# B&R Automation Studio project SiemensBRCommunication (part 2)

#### DAVclient.st - Services communcations between a B&R and Siemens PLC
```iecst
(********************************************************************************************************************************)
(* COPYRIGHT -- B&R Industrial Automation																																												*)
(********************************************************************************************************************************)
(* Library:				DAVNoDave																																																			*)
(* File: 					DAVclient.st																																																	*)
(* Author: 				morrisd																																																				*)
(* Created: 			June 02, 2009																																																	*)
(********************************************************************************************************************************)

(********************************************************************************************************************************)
(* DAVclient																																																										*)
(*==============================================================================================================================*)
(* Services communications between the PLC and the Siemen's PLC																																	*)
(* Returns a status																																																							*)
(********************************************************************************************************************************)
FUNCTION_BLOCK DAVclient

	(* Function not enabled *)
	IF(enable = FALSE)THEN
		status:= 65534;

	(* Invalid handle *)
	ELSIF(pHandle = 0)THEN
 		status:= DAV_ERR_HANDLE;

	(* Run the function *)
	ELSE
		(* Make status busy *)
		status:= 65535;

		(****************************************************************************************************************************)
		(* Initialize function																									                  																	*)
		(****************************************************************************************************************************)
		IF(state = 0)THEN
			pDAV ACCESS pHandle;																	(* Access handle *)

			(* Valid configuration 0 *)
			IF(pDAV.internal = 2)THEN
				pDAV.internal:= 3;

				(* Initialize DAVsend *)
				memset(ADR(DAVexchange_0), 0, SIZEOF(DAVexchange_0));
				DAVexchange_0.enable:=						TRUE;							(* Enable function block *)
				DAVexchange_0.pHandle:=						pHandle;					(* Handle from DAVinitialize *)
				DAVexchange_0.sendLength:=				0;								(* Size of sending data - calculated later *)
				DAVexchange_0.timeout:=						timeout;					(* Pass timeout *)
				DAVexchange_0.mpiFullExchange:=	 TRUE;							(* Enable full exchange of data *)

				(* Check initialization *)
				IF((pDAV.pBufferR <> 0) AND (pDAV.pBufferW <> 0) AND (pDAV.pConfig <> 0) AND (pDAV.pMapping <> 0) AND (pDAV.maxLinesMapping > 0))THEN

					(* Clear the internal variables *)
					IF(pDAV.maxLinesConfig > 0)THEN
						FOR itemIdx:=0 TO pDAV.maxLinesConfig-1 BY 1 DO
							pConfig ACCESS pDAV.pConfig + (itemIdx * SIZEOF(pConfig));
							pConfig.internal:= 0;
						END_FOR
					END_IF
					IF(pDAV.maxLinesMapping > 0)THEN
						FOR itemIdx:=0 TO pDAV.maxLinesMapping-1 BY 1 DO
							pMapping ACCESS pDAV.pMapping + (itemIdx * SIZEOF(pMapping));
							pMapping.internal:= 0;
						END_FOR
					END_IF
					itemIdx:= 0;																			(* Reset looping index *)
					state:= 2;																				(* Start function block - READ all WRITE data *)

				(* Connection closed *)
				ELSIF(pDAV.internal = 1)THEN
					status:= DAV_ERR_CONNECT_CLOSED;

				(* Critical error *)
				ELSE
					status:= DAV_ERR_INITIALIZATION;
				END_IF

			(* Critical error *)
			ELSE
				status:= DAV_ERR_INITIALIZATION;
			END_IF
		END_IF
		(****************************************************************************************************************************)

		(****************************************************************************************************************************)
		(* Request to initialize the client																																													*)
		(* Note: code placed underneath STATE 0, to ensure pDAV is a valid pointer																									*)
		(****************************************************************************************************************************)
		IF((pDAV.internal = 2) OR (
			(pDAV.connection.protocol <> DAV_PROTOCOL_TCP) AND (pDAV.connection.protocol <> DAV_PROTOCOL_MPI)) )THEN
			errorPackets:= 0;																			(* Clear number of error packets *)
			state:= 0;																						(* Reset function block *)
		END_IF
		(****************************************************************************************************************************)

		(****************************************************************************************************************************)
		(* Pause and Resume the function block                                                   																		*)
		(****************************************************************************************************************************)
		IF((pause = TRUE) AND (state = 1))THEN
			state:= 254;																					(* Pause function block *)
		END_IF
		IF((pause = FALSE) AND (state = 254))THEN
			state:= 1;																						(* Resume function block *)
		END_IF
		paused:= (state = 254);																	(* Show PAUSE status *)
		(****************************************************************************************************************************)

		(****************************************************************************************************************************)
		(* Completed reading all WRITE variables                                                																		*)
		(****************************************************************************************************************************)
		IF((state = 2) AND (itemIdx >= pDAV.maxLinesMapping))THEN

 			(* Clear the internal variables *)
			IF(pDAV.maxLinesConfig > 0)THEN
				FOR itemIdx:=0 TO pDAV.maxLinesConfig-1 BY 1 DO
					pConfig ACCESS pDAV.pConfig + (itemIdx * SIZEOF(pConfig));
					pConfig.internal:= 0;
				END_FOR
			END_IF

			(* Clear the internal variables *)
			IF(pDAV.maxLinesMapping > 0)THEN
				FOR itemIdx:=0 TO pDAV.maxLinesMapping-1 BY 1 DO
					pMapping ACCESS pDAV.pMapping + (itemIdx * SIZEOF(pMapping));
					pMapping.internal:= 0;
				END_FOR
			END_IF

			itemIdx:= 0;																					(* Reset looping index *)
			currentPriority:= 1;																	(* Reset the prioirty *)
			currentMode:= 0;																			(* Set mode to WRITE *)
			state:= 1;																						(* Run main routine *)
		END_IF
		(****************************************************************************************************************************)

		(****************************************************************************************************************************)
		(* Build up packet		                                                                  																		*)
		(****************************************************************************************************************************)
		IF(state = 1)THEN
			memset(pDAV.pBufferW, 0, DAV_DEFAULT_BUFFER_W);				(* Clear write buffer *)
			memset(ADR(varList), 0, SIZEOF(varList));							(* Clear list of variable index's *)
			numItems:= 0;																					(* Clear storage of our number of items *)
			numItemsCfg:= 0;																			(* Clear storage of our number of items *)
			numItemsMap:= 0;																			(* Clear storage of our number of items *)
			DAVexchange_0.sendLength:= 0;													(* Reset length to send *)

			(* Guesstimate the response length *)
			IF(pDAV.connection.protocol = DAV_PROTOCOL_TCP)THEN
				responseSize:= 21;																	(* Assume message type 3, with 2 byte parameter area *)
			ELSE
				responseSize:= 35;																	(* As above, but with BCC and assume some DLE doubling *)
			END_IF

			(* Repeat until we have data to send *)
			WHILE(state = 1)DO

				(************************************************************************************************************************)
				(* Initialize data																																																			*)
				(************************************************************************************************************************)

				(* WRITE mapping limit exceeded *)
				IF((currentMode = 0) AND (itemIdx >= pDAV.maxLinesMapping))THEN
					IF(pDAV.maxLinesConfig > 0)THEN
						currentMode:= 1;																(* Set mode to READ CONFIG *)
					ELSE
						currentMode:= 2;																(* Set mode to READ MAPPING*)
					END_IF
					itemIdx:= 0;																			(* Reset starting index *)

				(* READ config limit exceeded *)
				ELSIF((currentMode = 1) AND (itemIdx >= pDAV.maxLinesConfig))THEN
					currentMode:= 2;																	(* Set mode to READ MAPPING *)
					itemIdx:= 0;																			(* Reset starting index *)

				(* READ mapping limit exceeded *)
				ELSIF((currentMode = 2) AND (itemIdx >= pDAV.maxLinesMapping))THEN

		 			(* Clear the internal variables *)
					IF(pDAV.maxLinesConfig > 0)THEN
						FOR itemIdx:=0 TO pDAV.maxLinesConfig-1 BY 1 DO
							pConfig ACCESS pDAV.pConfig + (itemIdx * SIZEOF(pConfig));
							pConfig.internal:= 0;
						END_FOR
					END_IF

					(* Clear the internal variables *)
					IF(pDAV.maxLinesMapping > 0)THEN
						FOR itemIdx:=0 TO pDAV.maxLinesMapping-1 BY 1 DO
							pMapping ACCESS pDAV.pMapping + (itemIdx * SIZEOF(pMapping));
							pMapping.internal:= 0;
						END_FOR
					END_IF

	 				currentPriority:= (currentPriority MOD pDAV.maxPrioirty) + 1;		(* Increase the prioirty, reset to 1 *)
					currentMode:= 0;																	(* Set mode to WRITE *)
					itemIdx:= 0;																			(* Reset starting index *)
				END_IF
				(************************************************************************************************************************)

				(************************************************************************************************************************)
				(* Perform a write request 																																															*)
				(************************************************************************************************************************)
				IF(currentMode = 0)THEN
					memset(ADR(writeValues), 0, SIZEOF(writeValues));								(* Clear temp write values *)

					(* Determine the maximum size we can send *)
					IF(pDAV.connection.protocol = DAV_PROTOCOL_TCP)THEN
						maxSendSize:= DAV_PDU_SIZE - 20;								(* 12 byte parameter area, 8 byte data area with 4 byte variable *)
					ELSE
						maxSendSize:= DAV_PDU_SIZE - 30;								(* As above, but assume some DLE doubling *)
					END_IF

					(* Find WRITE requests *)
					FOR addIdx:= itemIdx TO pDAV.maxLinesMapping-1 BY 1 DO

						(* Access the current line (high prioirty or current priority) *)
						pMapping ACCESS pDAV.pMapping + (addIdx * SIZEOF(pMapping));

						(* Determine internal flags: *)
						(* "moreLinesToScan" - if we are still in the required priority *)
						(* "bufferFull" - if we have (or about to) reach the maximum limits imposed by the protocol *)
						moreLinesToScan:=	(pMapping.priority <= currentPriority);
						bufferFull:= (DAVexchange_0.sendLength > maxSendSize - pMapping.brVarLength) OR
													(responseSize >= DAV_PDU_SIZE - 1) OR (numItems >= 20);

						(* Cannot continue *)
						IF((bufferFull = TRUE) OR (moreLinesToScan = FALSE))THEN
							EXIT;

						(* W or R/W variables only *)
						ELSIF((pMapping.access = DAV_CONFIG_RW_W) OR (pMapping.access = DAV_CONFIG_RW_B))THEN

							(* Ensure variable is enabled *)
							IF(pMapping.pEnable > 0)THEN
			 					pEnable ACCESS pMapping.pEnable;
								useVariable:= (pEnable = TRUE);
							ELSE
								useVariable:= TRUE;
							END_IF

							(* Get the current value *)
							curValue:= 0;
							memcpy(ADR(curValue), pMapping.brVarAdr, pMapping.brVarLength);

							(* Packet should be added *)
							IF((useVariable = TRUE) AND (curValue <> pMapping.brPrevValue))THEN

								(* Initialise WRITE request *)
								IF(DAVexchange_0.sendLength = 0)THEN
					 				DAVexchange_0.sendLength:= DAVpacketWriteInit(pHandle, pDAV.pBufferW);
								END_IF

								(* Add variable to packet *)
								DAVexchange_0.sendLength:= DAVpacketWriteAddVar(pHandle, pDAV.pBufferW, pMapping.brVarAdr, ADR(pMapping.var));
								pMapping.internal:= 1;											(* Set variable in use *)
								responseSize:= responseSize + 1;						(* Increase estimate response size (16#FF) *)
								writeValues[numItems]:= curValue;						(* Store the value in our temporary buffer *)
								varList[numItems]:= addIdx;									(* Store variable index *)
								numItems:= numItems + 1;										(* Increase number of items *)

							(* Set WRITE variables to complete *)
							ELSIF((useVariable = FALSE) OR (pMapping.access = DAV_CONFIG_RW_W))THEN
								pMapping.internal:= 2;
							END_IF
						END_IF
					END_FOR

					(* No items found or limit reached *)
					IF((DAVexchange_0.sendLength = 0) OR (moreLinesToScan = FALSE) OR (addIdx >= pDAV.maxLinesMapping))THEN
						itemIdx:= pDAV.maxLinesMapping;									(* Force a reset on next loop iteration *)

					(* More lines remaining *)
					ELSE
						itemIdx:= addIdx;																(* Store the current index (for start of next scan) *)
					END_IF

					(* Now perform a WRITE request *)
					IF(DAVexchange_0.sendLength > 0)THEN

						(* Perform DLE doubling, DLE + ETX and BCC *)
						IF(pDAV.connection.protocol = DAV_PROTOCOL_MPI)THEN
							DAVexchange_0.sendLength:= DAVmpiSuffixCRC(pDAV.pBufferW, DAVexchange_0.sendLength);
						END_IF

						(* Continue *)
						state:= 10;
					END_IF
				(************************************************************************************************************************)

				(************************************************************************************************************************)
				(* Perform a read request 																																															*)
				(************************************************************************************************************************)
				ELSIF(currentMode = 1)THEN

					(* Config exists *)
					IF(pDAV.maxLinesConfig > 0)THEN

						(* Determine the maximum size we can send *)
						IF(pDAV.connection.protocol = DAV_PROTOCOL_TCP)THEN
							maxSendSize:= DAV_PDU_SIZE - 12;							(* 12 byte parameter area *)
						ELSE
							maxSendSize:= DAV_PDU_SIZE - 22;							(* As above, but assume some DLE doubling *)
						END_IF

						(* Find READ requests *)
						FOR addIdx:= itemIdx TO pDAV.maxLinesConfig-1 BY 1 DO

							(* Access the current line (high prioirty or current priority) *)
							pConfig ACCESS pDAV.pConfig + (addIdx * SIZEOF(pConfig));

							(* Determine internal flags: *)
							(* "moreLinesToScan" - if we are still in the required priority *)
							(* "bufferFull" - if we have (or about to) reach the maximum limits imposed by the protocol *)
							moreLinesToScan:=	(pMapping.priority <= currentPriority);
							bufferFull:= (DAVexchange_0.sendLength > maxSendSize) OR
														(responseSize > DAV_PDU_SIZE - 5 - pConfig.var.length) OR
														(numItems >= 20);

							(* Ensure variable is enabled *)
							IF(pConfig.pEnable > 0)THEN
			 					pEnable ACCESS pConfig.pEnable;
								useVariable:= (pEnable = TRUE);
							ELSE
								useVariable:= TRUE;
							END_IF

							(* Cannot continue *)
							IF((bufferFull = TRUE) OR (moreLinesToScan = FALSE))THEN
								EXIT;

							(* Variable not already used *)
							ELSIF((useVariable = TRUE) AND (pConfig.internal = 0))THEN

								(* Initialise READ request *)
								IF(DAVexchange_0.sendLength = 0)THEN
				 					DAVexchange_0.sendLength:= DAVpacketReadInit(pHandle, pDAV.pBufferW);
								END_IF

								(* Add variable to packet *)
								DAVexchange_0.sendLength:= DAVpacketReadAddVar(pHandle, pDAV.pBufferW, ADR(pConfig.var));
								pConfig.internal:= 1;												(* Set variable in use *)
								responseSize:= responseSize + 5 + pConfig.var.length;						(* Increase estimate response size *)
								varList[numItems]:= addIdx;									(* Store variable index *)
								numItems:= numItems + 1;										(* Increase number of items *)
								numItemsCfg:= numItemsCfg + 1;							(* Increase number of items *)
							END_IF
						END_FOR

						(* No items found or limit reached *)
						IF((DAVexchange_0.sendLength = 0) OR (moreLinesToScan = FALSE) OR (addIdx >= pDAV.maxLinesConfig))THEN
							itemIdx:= pDAV.maxLinesConfig;								(* Force a reset on next loop iteration *)

						(* More lines remaining - buffer full *)
						ELSE

							(* Perform DLE doubling, DLE + ETX and BCC *)
							IF(pDAV.connection.protocol = DAV_PROTOCOL_MPI)THEN
								DAVexchange_0.sendLength:= DAVmpiSuffixCRC(pDAV.pBufferW, DAVexchange_0.sendLength);
							END_IF

							(* Continue *)
							itemIdx:= addIdx;															(* Store the current index (for start of next scan) *)
							state:= 20;																		(* Send request now - no more data can be sent *)
						END_IF

					(* No Config *)
					ELSE
						currentMode:= 2;
					END_IF
				(************************************************************************************************************************)

				(************************************************************************************************************************)
				(* Perform a read request 																																															*)
				(************************************************************************************************************************)
				ELSE

					(* Determine the maximum size we can send *)
					IF(pDAV.connection.protocol = DAV_PROTOCOL_TCP)THEN
						maxSendSize:= DAV_PDU_SIZE - 12;								(* 12 byte parameter area *)
					ELSE
						maxSendSize:= DAV_PDU_SIZE - 22;								(* As above, but assume some DLE doubling *)
					END_IF

					(* Find READ requests *)
					FOR addIdx:= itemIdx TO pDAV.maxLinesMapping-1 BY 1 DO

						(* Access the current line (high prioirty or current priority) *)
						pMapping ACCESS pDAV.pMapping + (addIdx * SIZEOF(pMapping));

						(* Determine internal flags: *)
						(* "moreLinesToScan" - if we are still in the required priority *)
						(* "bufferFull" - if we have (or about to) reach the maximum limits imposed by the protocol *)
						moreLinesToScan:=	(pMapping.priority <= currentPriority);
						bufferFull:= (DAVexchange_0.sendLength > maxSendSize) OR
													(responseSize > DAV_PDU_SIZE - 5 - pMapping.brVarLength) OR
													(numItems >= 20);

						(* Cannot continue *)
						IF((bufferFull = TRUE) OR (moreLinesToScan = FALSE))THEN
							EXIT;

						(* Variable not already used *)
						ELSIF(pMapping.internal = 0)THEN

							(* READ request already contains configuration items *)
							IF((numItemsCfg > 0) AND (pMapping.cfgIndex < 65535) AND (pMapping.cfgIndex < pDAV.maxLinesConfig))THEN
			 					pConfig ACCESS pDAV.pConfig + (pMapping.cfgIndex * SIZEOF(pConfig));
								useVariable:= (pConfig.internal <> 1);						(* Use variable if the config is not currently in use *)
							ELSE
								useVariable:= TRUE;
							END_IF

							(* Ensure variable is enabled *)
							IF(pMapping.pEnable > 0)THEN
			 					pEnable ACCESS pMapping.pEnable;
								useVariable:= useVariable AND (pEnable = TRUE);

								(* Set variable used if it is disabled *)
								IF(pEnable = FALSE)THEN
									pMapping.internal:= 2;
								END_IF
							END_IF

							(* Variable can be added *)
							IF(useVariable = TRUE)THEN

								(* Initialise READ request *)
								IF(DAVexchange_0.sendLength = 0)THEN
				 					DAVexchange_0.sendLength:= DAVpacketReadInit(pHandle, pDAV.pBufferW);
								END_IF

								(* Add variable to packet *)
								DAVexchange_0.sendLength:= DAVpacketReadAddVar(pHandle, pDAV.pBufferW, ADR(pMapping.var));
								pMapping.internal:= 1;											(* Set variable in use *)
								responseSize:= responseSize + 5 + pMapping.brVarLength;				(* Increase estimate response size *)
								varList[numItems]:= addIdx;									(* Store variable index *)
								numItems:= numItems + 1;										(* Increase number of items *)
								numItemsMap:= numItemsMap + 1;							(* Increase number of items *)
							END_IF
						END_IF
					END_FOR

					(* No items found or limit reached *)
					IF((DAVexchange_0.sendLength = 0) OR (moreLinesToScan = FALSE) OR (addIdx >= pDAV.maxLinesMapping))THEN
						itemIdx:= pDAV.maxLinesMapping;									(* Force a reset on next loop iteration *)

					(* More lines remaining - buffer full *)
					ELSE
						itemIdx:= addIdx;																(* Store the current index (for start of next scan) *)
					END_IF

					(* Now perform a READ request *)
					IF(DAVexchange_0.sendLength > 0)THEN

						(* Perform DLE doubling, DLE + ETX and BCC *)
						IF(pDAV.connection.protocol = DAV_PROTOCOL_MPI)THEN
							DAVexchange_0.sendLength:= DAVmpiSuffixCRC(pDAV.pBufferW, DAVexchange_0.sendLength);
						END_IF

						(* Continue *)
						state:= 20;

					(* No data to send, exit loop to avoid a cycle time violation *)
					ELSE
						EXIT;
					END_IF
				END_IF
				(************************************************************************************************************************)
			END_WHILE
		(****************************************************************************************************************************)

		(****************************************************************************************************************************)
		(* Build up packet READ WRITE data first                                                																		*)
		(****************************************************************************************************************************)
		ELSIF(state = 2)THEN
			memset(pDAV.pBufferW, 0, DAV_DEFAULT_BUFFER_W);				(* Clear write buffer *)
			memset(ADR(varList), 0, SIZEOF(varList));							(* Clear list of variable index's *)
			numItems:= 0;																					(* Clear storage of our number of items *)
			numItemsCfg:= 0;																			(* Clear storage of our number of items *)
			numItemsMap:= 0;																			(* Clear storage of our number of items *)
			DAVexchange_0.sendLength:= 0;													(* Reset length to send *)

			(* Guesstimate the response length *)
			IF(pDAV.connection.protocol = DAV_PROTOCOL_TCP)THEN
				responseSize:= 21;																	(* Assume message type 3, with 2 byte parameter area *)
				maxSendSize:= DAV_PDU_SIZE - 12;										(* 12 byte parameter area *)
			ELSE
				responseSize:= 35;																	(* As above, but with BCC and assume some DLE doubling *)
				maxSendSize:= DAV_PDU_SIZE - 22;										(* As above, but assume some DLE doubling *)
			END_IF

			(**************************************************************************************************************************)
			(* Perform a read request 																																																*)
			(**************************************************************************************************************************)
			FOR addIdx:= itemIdx TO pDAV.maxLinesMapping-1 BY 1 DO

				(* Access the current line (high prioirty or current priority) *)
				pMapping ACCESS pDAV.pMapping + (addIdx * SIZEOF(pMapping));

				(* Determine internal flags: *)
				(* "bufferFull" - if we have (or about to) reach the maximum limits imposed by the protocol *)
				bufferFull:= (DAVexchange_0.sendLength > maxSendSize) OR
											(responseSize > DAV_PDU_SIZE - 5 - pMapping.brVarLength) OR
											(numItems >= 20);

				(* Cannot continue *)
				IF(bufferFull = TRUE)THEN
					EXIT;

				(* Variable not already used *)
				ELSIF((pMapping.access <> DAV_CONFIG_RW_R) AND (pMapping.internal = 0))THEN

					(* Initialise READ request *)
					IF(DAVexchange_0.sendLength = 0)THEN
	 					DAVexchange_0.sendLength:= DAVpacketReadInit(pHandle, pDAV.pBufferW);
					END_IF

					(* Add variable to packet *)
					DAVexchange_0.sendLength:= DAVpacketReadAddVar(pHandle, pDAV.pBufferW, ADR(pMapping.var));
					pMapping.internal:= 1;													(* Set variable in use *)
					responseSize:= responseSize + 5 + pMapping.brVarLength;				(* Increase estimate response size *)
					varList[numItems]:= addIdx;											(* Store variable index *)
					numItems:= numItems + 1;												(* Increase number of items *)
					numItemsMap:= numItemsMap + 1;									(* Increase number of items *)
				END_IF
			END_FOR

			(* No items found or limit reached *)
			IF((DAVexchange_0.sendLength = 0) OR (addIdx >= pDAV.maxLinesMapping))THEN
				itemIdx:= pDAV.maxLinesMapping;										(* Force a reset on next loop iteration *)

			(* More lines remaining - buffer full *)
			ELSE
				itemIdx:= addIdx;																	(* Store the current index (for start of next scan) *)
			END_IF

			(* Now perform a READ request *)
			IF(DAVexchange_0.sendLength > 0)THEN

				(* Perform DLE doubling, DLE + ETX and BCC *)
				IF(pDAV.connection.protocol = DAV_PROTOCOL_MPI)THEN
					DAVexchange_0.sendLength:= DAVmpiSuffixCRC(pDAV.pBufferW, DAVexchange_0.sendLength);
				END_IF

				(* Continue *)
				state:= 30;
			END_IF
		END_IF
		(****************************************************************************************************************************)

		(****************************************************************************************************************************)
		(* Function Operation (R/W)                                                                																	*)
		(****************************************************************************************************************************)
		CASE state OF

			(**************************************************************************************************************************)
			(* Send a WRITE command																								                  																	*)
			(**************************************************************************************************************************)
			10:
				(* Service function *)
				DAVexchange_0();

				(* Data sent and received *)
				IF(DAVexchange_0.status = 0)THEN

					(* Access buffer *)
					ppBuffer ACCESS pDAV.pBufferR + DAVexchange_0.recvStartOfDataIdx;

					(* Ensure we have received a WRITE packet and the correct number of items *)
					IF((ppBuffer[0] = 16#05) AND (ppBuffer[1] = numItems) AND
						(DAVexchange_0.recvParamLength = 2) AND (DAVexchange_0.recvDataLength = numItems))THEN

						(* Re-access buffer *)
						ppBuffer ACCESS pDAV.pBufferR + DAVexchange_0.recvStartOfDataIdx + DAVexchange_0.recvParamLength;

						(* Store the value of each variable if it is successfull *)
						FOR findIdx:=0 TO numItems-1 BY 1 DO

							(* Access the current line *)
							pMapping ACCESS pDAV.pMapping + (varList[findIdx] * SIZEOF(pMapping));

							(* Found an item in use *)
							IF(pMapping.internal = 1)THEN

								(* Parameter has been written succesfully, copy data into variable's previous value *)
								IF(ppBuffer[findIdx] = 16#FF)THEN
									pMapping.brPrevValue:= writeValues[findIdx];

								(* Invalid reponse *)
								ELSE
									status:= DAV_ERR_FAILED_WRITE;
									errorPackets:= errorPackets + 1;
								END_IF
								pMapping.internal:= 2;										(* Set variable completed *)
							END_IF
						END_FOR

					(* Wrong packet received *)
					ELSE
						status:= DAV_ERR_RECV_WRONGPACKET;
						errorPackets:= errorPackets + 1;
					END_IF

					state:= 1;																			(* Return to the running state *)

				(* Error *)
				ELSIF(DAVexchange_0.status <> 65535)THEN
					status:= DAVexchange_0.status;
					state:= 0;
				END_IF
			(**************************************************************************************************************************)

			(**************************************************************************************************************************)
			(* Send a READ command																								                  																	*)
			(**************************************************************************************************************************)
			20:
				(* Service function *)
				DAVexchange_0();

				(* Data sent and received *)
				IF(DAVexchange_0.status = 0)THEN

					(* Access buffer *)
					ppBuffer ACCESS pDAV.pBufferR + DAVexchange_0.recvStartOfDataIdx;

					(* Ensure we have received a READ packet and the correct number of items *)
					IF((ppBuffer[0] = 16#04) AND (ppBuffer[1] = numItems) AND
						(DAVexchange_0.recvParamLength = 2) AND (DAVexchange_0.recvDataLength > 0))THEN

						(* Re-access buffer *)
						ppBuffer ACCESS pDAV.pBufferR + DAVexchange_0.recvStartOfDataIdx + DAVexchange_0.recvParamLength;
						readIdx:= 0;

						(*------------------------------------------------------------------------------------------------------------------*)
						(* Store the value of each variable if it is successfull 																														*)
						(*------------------------------------------------------------------------------------------------------------------*)
						IF(numItemsCfg > 0)THEN
							FOR findIdx:=0 TO numItemsCfg-1 BY 1 DO
								pConfig ACCESS pDAV.pConfig + (varList[findIdx] * SIZEOF(pConfig));

								(* Found an item in use *)
								IF(pConfig.internal = 1)THEN

									(* Parameter has been read succesfully - BOOL *)
									IF((ppBuffer[readIdx] = 16#FF) AND (ppBuffer[readIdx+1] = 16#03))THEN
										dataLength:= DAVswapWORD(ADR(ppBuffer[readIdx+2]));				(* Get datalength as bytes *)

									(* Parameter has been read succesfully - BYTE *)
									ELSIF((ppBuffer[readIdx] = 16#FF) AND (ppBuffer[readIdx+1] = 16#04))THEN
										dataLength:= DAVswapWORD(ADR(ppBuffer[readIdx+2])) / 8;		(* Get datalength as bytes *)

									(* Error *)
									ELSE
										dataLength:= 0;
										errorPackets:= errorPackets + 1;
									END_IF

									(* Check length is the same and copy *)
									IF((dataLength > 0) AND (dataLength = pConfig.var.length))THEN
										memcpy(pConfig.brVarAdr, ADR(ppBuffer[readIdx+4]), pConfig.var.length);		(* Copy data into memory block *)

										(* Now map this data using the mapping congifuration *
										FOR mapIdx:=0 TO pDAV.maxLinesMapping-1 BY 1 DO
											pMapping ACCESS pDAV.pMapping + (mapIdx * SIZEOF(pMapping));

											(* Ensure variable is enabled *
											IF(pMapping.pEnable > 0)THEN
			 									pEnable ACCESS pMapping.pEnable;
												useVariable:= (pEnable = TRUE);
											ELSE
												useVariable:= TRUE;
											END_IF

											(* Uses a custom mapping - update it *
											DAVcalcVARadr(ADR(pMapping.var));

											IF((useVariable = TRUE) AND
												(pMapping.access < DAV_CONFIG_RW_W) AND
												(pMapping.var.area = pConfig.var.area) AND
												(pMapping.var.db = pConfig.var.db) AND
												(pMapping.var.bitAdr >= pConfig.var.bitAdr) AND
												(pMapping.var.bitAdr + SEL((pMapping.var.type = DAV_VAR_BIT), (pMapping.var.length * 8), 1) <=
												 	pConfig.var.bitAdr + SEL((pConfig.var.type = DAV_VAR_BIT), (pConfig.var.length * 8), 1)))THEN

												(* R/W variable - check if the value has changed *
												IF(pMapping.access = DAV_CONFIG_RW_B)THEN
													curValue:= 0;
													memcpy(ADR(curValue), pMapping.brVarAdr, pMapping.brVarLength);
												END_IF

												(* Packet should be updated *
												IF((pMapping.access = DAV_CONFIG_RW_R) OR
												((pMapping.access = DAV_CONFIG_RW_B) AND (curValue = pMapping.brPrevValue)))THEN
													(*DAVupdateVAR(ADR(pMapping), pConfig.brVarAdr + pMapping.var.actAdr - pConfig.var.actAdr);*
													DAVupdateVAR(ADR(pMapping), pConfig.brVarAdr + (
													((pMapping.var.bitAdr AND 16#FFF8) - pConfig.var.bitAdr) / 8), FALSE);
													pMapping.internal:= 2;
												END_IF
											END_IF
										END_FOR

									(* Error *)
									ELSE
										status:= DAV_ERR_FAILED_READ;
										errorPackets:= errorPackets + 1;
									END_IF

									readIdx:= readIdx + 4 + dataLength + (dataLength MOD 2);		(* Next offset (2 byte allignment) *)
									pConfig.internal:= 3;											(* Set variable completed *)
								END_IF
							END_FOR

							(* Now map this data using the mapping congifuration *)
							FOR mapIdx:=0 TO pDAV.maxLinesMapping-1 BY 1 DO
								pMapping ACCESS pDAV.pMapping + (mapIdx * SIZEOF(pMapping));

								(* Uses a configuration *)
								IF(pMapping.cfgIndex <> 65535)THEN
									pConfig ACCESS pDAV.pConfig + (pMapping.cfgIndex * SIZEOF(pConfig));

									(* Ensure variable is enabled *)
									useVariable:= (pConfig.internal = 3);
									IF((useVariable = TRUE) AND (pMapping.pEnable > 0))THEN
 										pEnable ACCESS pMapping.pEnable;
										useVariable:= (pEnable = TRUE);
									END_IF

									(* Variable can be updated *)
									IF(useVariable = TRUE)THEN

										(* Uses a custom mapping - update it *)
										DAVcalcVARadr(ADR(pMapping.var));

										IF((pMapping.access < DAV_CONFIG_RW_W) AND
											(pMapping.var.area = pConfig.var.area) AND
											(pMapping.var.db = pConfig.var.db) AND
											(pMapping.var.bitAdr >= pConfig.var.bitAdr) AND
											(pMapping.var.bitAdr + SEL((pMapping.var.type = DAV_VAR_BIT), (pMapping.var.length * 8), 1) <=
											 	pConfig.var.bitAdr + SEL((pConfig.var.type = DAV_VAR_BIT), (pConfig.var.length * 8), 1)))THEN

											(* R/W variable - check if the value has changed *)
											IF(pMapping.access = DAV_CONFIG_RW_B)THEN
												curValue:= 0;
												memcpy(ADR(curValue), pMapping.brVarAdr, pMapping.brVarLength);
											END_IF

											(* Packet should be updated *)
											IF((pMapping.access = DAV_CONFIG_RW_R) OR
											((pMapping.access = DAV_CONFIG_RW_B) AND (curValue = pMapping.brPrevValue)))THEN

												DAVupdateVAR(ADR(pMapping), pConfig.brVarAdr + (
												((pMapping.var.bitAdr AND 16#FFF8) - pConfig.var.bitAdr) / 8), FALSE);
												pMapping.internal:= 2;
											END_IF
										END_IF
									END_IF
								END_IF
							END_FOR

							(* Set internal to complete *)
							FOR findIdx:=0 TO numItemsCfg-1 BY 1 DO
								pConfig ACCESS pDAV.pConfig + (findIdx * SIZEOF(pConfig));

								IF(pConfig.internal = 3)THEN
					 				pConfig.internal:= 2;
								END_IF
							END_FOR
						END_IF
						(*------------------------------------------------------------------------------------------------------------------*)

						(*------------------------------------------------------------------------------------------------------------------*)
						(* Store the value of each variable if it is successfull 																														*)
						(*------------------------------------------------------------------------------------------------------------------*)
						IF(numItemsMap > 0)THEN
							FOR findIdx:=0 TO numItemsMap-1 BY 1 DO
								pMapping ACCESS pDAV.pMapping + (varList[numItemsCfg + findIdx] * SIZEOF(pMapping));

								(* Found an item in use *)
								IF(pMapping.internal = 1)THEN

									(* Parameter has been read succesfully - BOOL *)
									IF((ppBuffer[readIdx] = 16#FF) AND (ppBuffer[readIdx+1] = 16#03))THEN
										dataLength:= DAVswapWORD(ADR(ppBuffer[readIdx+2]));				(* Get datalength as bytes *)

									(* Parameter has been read succesfully - BYTE *)
									ELSIF((ppBuffer[readIdx] = 16#FF) AND (ppBuffer[readIdx+1] = 16#04))THEN
										dataLength:= DAVswapWORD(ADR(ppBuffer[readIdx+2])) / 8;		(* Get datalength as bytes *)

									(* Error *)
									ELSE
										dataLength:= 0;
										errorPackets:= errorPackets + 1;
									END_IF

									(* Check length is the same and copy *)
									IF((dataLength > 0) AND (dataLength = pMapping.var.length))THEN

										(* R/W variable - check if the value has changed *)
										IF(pMapping.access = DAV_CONFIG_RW_B)THEN
											curValue:= 0;
											memcpy(ADR(curValue), pMapping.brVarAdr, pMapping.brVarLength);
										END_IF

										(* Packet should be updated *)
										IF((pMapping.access = DAV_CONFIG_RW_R) OR (curValue = pMapping.brPrevValue))THEN
											DAVupdateVAR(ADR(pMapping), ADR(ppBuffer[readIdx+4]), (ppBuffer[readIdx+1] = 16#03));
										END_IF

									(* Error *)
									ELSE
										status:= DAV_ERR_FAILED_READ;
										errorPackets:= errorPackets + 1;
									END_IF
									pMapping.internal:= 2;
								END_IF
								readIdx:= readIdx + 4 + dataLength + (dataLength MOD 2);		(* Next offset (2 byte allignment) *)
							END_FOR
						END_IF
						(*------------------------------------------------------------------------------------------------------------------*)

					(* Wrong packet received *)
					ELSE
						status:= DAV_ERR_RECV_WRONGPACKET;
						errorPackets:= errorPackets + 1;
					END_IF
					state:= 1;																			(* Return to the running state *)

				(* Error *)
				ELSIF(DAVexchange_0.status <> 65535)THEN
					status:= DAVexchange_0.status;
					state:= 0;
				END_IF
			(**************************************************************************************************************************)

			(**************************************************************************************************************************)
			(* Send a READ command (for WRITE data)																                  																	*)
			(**************************************************************************************************************************)
			30:
				(* Service function *)
				DAVexchange_0();

				(* Data sent and received *)
				IF(DAVexchange_0.status = 0)THEN

					(* Access buffer *)
					ppBuffer ACCESS pDAV.pBufferR + DAVexchange_0.recvStartOfDataIdx;

					(* Ensure we have received a READ packet and the correct number of items *)
					IF((ppBuffer[0] = 16#04) AND (ppBuffer[1] = numItems) AND
						(DAVexchange_0.recvParamLength = 2) AND (DAVexchange_0.recvDataLength > 0))THEN

						(* Re-access buffer *)
						ppBuffer ACCESS pDAV.pBufferR + DAVexchange_0.recvStartOfDataIdx + DAVexchange_0.recvParamLength;
						readIdx:= 0;

						(*------------------------------------------------------------------------------------------------------------------*)
						(* Store the value of each variable if it is successfull 																														*)
						(*------------------------------------------------------------------------------------------------------------------*)
						IF(numItemsMap > 0)THEN
							FOR findIdx:=0 TO numItemsMap-1 BY 1 DO
								pMapping ACCESS pDAV.pMapping + (varList[numItemsCfg + findIdx] * SIZEOF(pMapping));

								(* Found an item in use *)
								IF(pMapping.internal = 1)THEN

									(* Parameter has been read succesfully - BOOL *)
									IF((ppBuffer[readIdx] = 16#FF) AND (ppBuffer[readIdx+1] = 16#03))THEN
										dataLength:= DAVswapWORD(ADR(ppBuffer[readIdx+2]));				(* Get datalength as bytes *)

									(* Parameter has been read succesfully - BYTE *)
									ELSIF((ppBuffer[readIdx] = 16#FF) AND (ppBuffer[readIdx+1] = 16#04))THEN
										dataLength:= DAVswapWORD(ADR(ppBuffer[readIdx+2])) / 8;		(* Get datalength as bytes *)

									(* Error *)
									ELSE
										dataLength:= 0;
										errorPackets:= errorPackets + 1;
									END_IF

									(* Check length is the same and copy *)
									IF((dataLength > 0) AND (dataLength = pMapping.var.length))THEN

										(* Update variable *)
										DAVupdateVAR(ADR(pMapping), ADR(ppBuffer[readIdx+4]), (ppBuffer[readIdx+1] = 16#03));

									(* Error *)
									ELSE
										status:= DAV_ERR_FAILED_READ;
										errorPackets:= errorPackets + 1;
									END_IF
									pMapping.internal:= 2;
								END_IF
								readIdx:= readIdx + 4 + dataLength + (dataLength MOD 2);		(* Next offset (2 byte allignment) *)
							END_FOR
						END_IF
						(*------------------------------------------------------------------------------------------------------------------*)

					(* Wrong packet received *)
					ELSE
						status:= DAV_ERR_RECV_WRONGPACKET;
						errorPackets:= errorPackets + 1;
					END_IF
					state:= 2;																			(* Return to the running state *)

				(* Error *)
				ELSIF(DAVexchange_0.status <> 65535)THEN
					status:= DAVexchange_0.status;
				END_IF
			(**************************************************************************************************************************)

		END_CASE
		(****************************************************************************************************************************)
		(* End of Function Operation                                                             																		*)
		(****************************************************************************************************************************)
	END_IF

	(******************************************************************************************************************************)
	(* Reset to state 0 when in error																																															*)
	(******************************************************************************************************************************)
	IF(status <> 65535)THEN
		state:= 0;
	END_IF
	(******************************************************************************************************************************)

	(******************************************************************************************************************************)
	(* Update when it is safe to disconnect																																												*)
	(******************************************************************************************************************************)
	safeToDisconnect:= (state = 1);
	(******************************************************************************************************************************)

END_FUNCTION_BLOCK
(********************************************************************************************************************************)
(* End of DAVclient																																																							*)
(********************************************************************************************************************************)
```

#### DAVexchange.st - Exchanges data between PLC's
```iecst
(********************************************************************************************************************************)
(* COPYRIGHT -- B&R Industrial Automation																																												*)
(********************************************************************************************************************************)
(* Library:				DAVNoDave																																																			*)
(* File: 					DAVexchange.st																																																*)
(* Author: 				morrisd																																																				*)
(* Created: 			May 26, 2009																																																	*)
(********************************************************************************************************************************)

(********************************************************************************************************************************)
(* DAVexchange																																																									*)
(*==============================================================================================================================*)
(* Sends a packet to the PLC									 																																									*)
(* Receives the response from the PLC 																																													*)
(* Returns a status																																																							*)
(********************************************************************************************************************************)
FUNCTION_BLOCK DAVexchange

	(* Function not enabled *)
	IF(enable = FALSE)THEN
		status:= 65534;

	(* Invalid handle *)
	ELSIF(pHandle = 0)THEN
 		status:= DAV_ERR_HANDLE;

	(* Invalid buffer length *)
	ELSIF((sendLength = 0) OR (sendLength > DAV_DEFAULT_BUFFER_W))THEN
 		status:= DAV_ERR_BUFFER_SIZE;

	(* Run the function *)
	ELSE

		(* Make status busy *)
		status:= 65535;

		(****************************************************************************************************************************)
		(* Map data (to avoid errors if the user changes them during operation                  																		*)
		(* Note: code placed here to avoid a 1 scan delay																																						*)
		(****************************************************************************************************************************)
		IF(state = 0)THEN

			(* Reset received number of bytes *)
			recvLength:= 					0;
			recvParamLength:= 		0;
			recvDataLength:= 			0;
			recvStartOfDataIdx:=	0;

			(* Access handle *)
			pDAV ACCESS pHandle;

			(* Access buffer *)
			ppBuffer ACCESS pDAV.pBufferR;
			memset(pDAV.pBufferR, 0, DAV_DEFAULT_BUFFER_R);

			(* Initialize TON timeout function block *)
			TON_10ms_Timeout.IN:=					FALSE;									(* Turn timer off *)
			IF((timeout = 0) AND (pDAV.connection.protocol = DAV_PROTOCOL_TCP))THEN
				TON_10ms_Timeout.PT:=				150;										(* Default TCP tiemout = 1.5s *)
			ELSIF(timeout = 0)THEN
				TON_10ms_Timeout.PT:=				500;										(* Default MPI tiemout = 5s *)
			ELSE
				TON_10ms_Timeout.PT:= 			timeout;								(* User's timeout *)
			END_IF
			TON_10ms_Timeout();																		(* Call function to reset timer *)
			TON_10ms_Timeout.IN:= 				TRUE;										(* Enable timer *)

			(* Initialize TCP coms *)
			IF(pDAV.connection.protocol = DAV_PROTOCOL_TCP)THEN

				(* Initialize TcpSend function block *)
				TcpSend_0.enable:=					TRUE;										(* Enable function block *)
				TcpSend_0.ident:=						pDAV.ident;							(* TcpOpen ident *)
				TcpSend_0.pData:=						pDAV.pBufferW;					(* Address of write buffer *)
				TcpSend_0.datalen:=					sendLength;							(* Length of data to send *)
				TcpSend_0.flags:=						0;											(* Default options *)

				(* Initialize TcpSend function block *)
				TcpRecv_0.enable:=					TRUE;										(* Enable function block *)
				TcpRecv_0.ident:=						pDAV.ident;							(* TcpOpen ident *)
				TcpRecv_0.pData:=						pDAV.pBufferR;					(* Address of read buffer *)
				TcpRecv_0.datamax:=				 	DAV_DEFAULT_BUFFER_R;		(* Size of read buffer *)
				TcpRecv_0.flags:= 					0;											(* Default options *)

				(* Go to next state *)
				state:= 100;

			(* Initialize MPI coms *)
			ELSIF(pDAV.connection.protocol = DAV_PROTOCOL_MPI)THEN

				(* Initialize DAVmpiSend function block *)
				DAVmpiSend_0.enable:=				TRUE;										(* Enable function block *)
				DAVmpiSend_0.ident:=				pDAV.ident;							(* FRM_Xopen ident *)
				DAVmpiSend_0.pBufferW:=			ADR(bufferSend);				(* Default to internal buffer *)
				DAVmpiSend_0.sendLength:=		0;											(* Clear send length (will change) *)

				(* Initialize DAVmpiRead function block *)
				DAVmpiRead_0.enable:=				TRUE;										(* Enable function block *)
				DAVmpiRead_0.ident:=				pDAV.ident;							(* FRM_Xopen ident *)
				DAVmpiRead_0.pBufferR:=			ADR(bufferRead);				(* Default to internal buffer *)
				DAVmpiRead_0.readLength:=		SIZEOF(bufferRead);			(* Size of read buffer *)

				(* Clear buffers *)
				memset(ADR(bufferSend), 0, SIZEOF(bufferSend));
				memset(ADR(bufferRead), 0, SIZEOF(bufferRead));

				(* Initialize STATE 200 *)
				bufferSend[0]:=							16#02;									(* STX *)
				DAVmpiSend_0.sendLength:=		1;											(* Length to send *)

				(* Go to next state *)
				state:= 200;

			(* Invalid mode *)
			ELSE
				status:= DAV_ERR_CONNECT_PROTOCOL;
			END_IF
		END_IF
		(****************************************************************************************************************************)

		(****************************************************************************************************************************)
		(* Function Operation                                                                     																	*)
		(****************************************************************************************************************************)
		CASE state OF

			(**************************************************************************************************************************)
			(* TCP Write - message                                                                   																	*)
			(**************************************************************************************************************************)
			100:
				(* Service function *)
				TcpSend_0();

				(* Data sent *)
				IF((TcpSend_0.status = 0) AND (TcpSend_0.sentlen = TcpSend_0.datalen))THEN
		 				state:= 101;

				(* Not all the data was sent *)
				ELSIF(TcpSend_0.status = 0)THEN
					status:= DAV_ERR_SEND_MISSINGDATA;

				(* Error *)
				ELSIF(TcpSend_0.status <> 65535)THEN
					status:= TcpSend_0.status;
				END_IF
			(**************************************************************************************************************************)

			(**************************************************************************************************************************)
			(* TCP Read - message                                                                    																	*)
			(**************************************************************************************************************************)
			101:
				(* Service function *)
				TcpRecv_0();

				(* Service timeout *)
				TON_10ms_Timeout();

				(* Data received *)
				IF((TcpRecv_0.status = 0) AND (TcpRecv_0.recvlen > 0))THEN
					recvLength:= DAVswapWORD(ADR(ppBuffer[2]));								(* Bytes ppBuffer[2] and [3] *)

					(* Not all the data has been received *)
					IF(recvLength <> UDINT_TO_UINT(TcpRecv_0.recvlen))THEN
				 		recvLength:= UDINT_TO_UINT(TcpRecv_0.recvlen);
				 		status:= DAV_ERR_RECV_MISSINGDATA;

				 	(* Complete *)
				 	ELSE
						(* Return Parameter and Data lengths *)
						recvParamLength:= DAVswapWORD(ADR(ppBuffer[13]));				(* Bytes ppBuffer[13] and [14] *)
						recvDataLength:= DAVswapWORD(ADR(ppBuffer[15]));				(* Bytes ppBuffer[15] and [16] *)

						(* Return the start of the data index *)
						IF((ppBuffer[8] = 2) OR (ppBuffer[8] = 3))THEN
							recvStartOfDataIdx:= 19; (*7 + 12;*)
						ELSE
							recvStartOfDataIdx:= 17; (*7 + 10;*)
						END_IF

						(* Reduce receive length for length of data *)
						IF(recvLength >= recvStartOfDataIdx)THEN
		 					recvLength:= recvLength - recvStartOfDataIdx;
						ELSE
							recvLength:= 0;
						END_IF
						status:= 0;
					END_IF

				(* Invalid receive length *)
				ELSIF(TcpRecv_0.status = 0)THEN
					status:= DAV_ERR_RECV_NODATA;

				(* Timeout *)
				ELSIF(TON_10ms_Timeout.Q)THEN
					status:= DAV_ERR_TIMEOUT;

				(* No data - try again *)
				ELSIF(TcpRecv_0.status = tcpERR_NO_DATA)THEN
					state:= state;

				(* Error *)
				ELSIF(TcpRecv_0.status <> 65535)THEN
					status:= TcpRecv_0.status;
				END_IF
			(**************************************************************************************************************************)

			(**************************************************************************************************************************)
			(* MPI Write - STX		                                                                   																	*)
			(**************************************************************************************************************************)
			200:
				(* Service function *)
				DAVmpiSend_0();

				(* Data written *)
				IF(DAVmpiSend_0.status = 0)THEN
			 		bufferSend[0]:= 0;
					state:= 201;

				(* Error writing data *)
				ELSIF(DAVmpiSend_0.status <> 65535)THEN
					status:= DAVmpiSend_0.status;
				END_IF
			(**************************************************************************************************************************)

			(**************************************************************************************************************************)
			(* MPI Read - DLE                                                               																					*)
			(**************************************************************************************************************************)
			201:
				(* Service function *)
        DAVmpiRead_0();

				(* Service timeout *)
				TON_10ms_Timeout();

				(* Data received - DLE *)
				IF((DAVmpiRead_0.status = 0) AND (DAVmpiRead_0.recvBufferLength = 1) AND (bufferRead[0] = 16#10))THEN

					(* Reset timer *)
					TON_10ms_Timeout.IN:= FALSE;
					TON_10ms_Timeout();
					TON_10ms_Timeout.IN:= TRUE;

					(* Point to the message buffer *)
					DAVmpiSend_0.pBufferW:=			pDAV.pBufferW;
					DAVmpiSend_0.sendLength:=		sendLength;

					(* Continue *)
					bufferRead[0]:= 0;
					state:= 202;

				(* Invalid data *)
				ELSIF(DAVmpiRead_0.status = 0)THEN
					status:= DAV_ERR_RECV_PROTOCOL;

				(* Timeout *)
				ELSIF(TON_10ms_Timeout.Q)THEN
					status:= DAV_ERR_TIMEOUT;

				(* Error *)
				ELSIF(DAVmpiRead_0.status <> 65535)THEN
					status:= DAVmpiRead_0.status;
				END_IF
			(**************************************************************************************************************************)

			(**************************************************************************************************************************)
			(* MPI Write - message                                                                   																	*)
			(**************************************************************************************************************************)
			202:
				(* Service function *)
				DAVmpiSend_0();

				(* Data written *)
				IF(DAVmpiSend_0.status = 0)THEN

					(* Point to the internal buffer *)
					DAVmpiSend_0.pBufferW:= ADR(bufferSend);
			 		state:= 203;

				(* Error writing data *)
				ELSIF(DAVmpiSend_0.status <> 65535)THEN
					status:= DAVmpiSend_0.status;
				END_IF
			(**************************************************************************************************************************)

			(**************************************************************************************************************************)
			(* MPI Read - DLE | DLE + STX                                                    																					*)
			(**************************************************************************************************************************)
			203:
				(* Service function *)
        DAVmpiRead_0();

				(* Service timeout *)
				TON_10ms_Timeout();

				(* Data received *)
				IF((DAVmpiRead_0.status = 0) AND (
					((DAVmpiRead_0.recvBufferLength = 2) AND (bufferRead[0] = 16#10) AND (bufferRead[1] = 16#02)) OR
					((DAVmpiRead_0.recvBufferLength = 1) AND (bufferRead[0] = 16#10)) ))THEN

					(* Reset timer *)
					TON_10ms_Timeout.IN:= FALSE;
					TON_10ms_Timeout();
					TON_10ms_Timeout.IN:= TRUE;

		 			(* Valid data - DLE STX *)
					bufferRead[0]:= 0;
					IF(DAVmpiRead_0.recvBufferLength = 2)THEN
						bufferRead[1]:= 0;
		 				state:= 205;

					(* Valid data - DLE *)
					ELSE
						state:= 204;
					END_IF

				(* Invalid protocol *)
				ELSIF(DAVmpiRead_0.status = 0)THEN
					status:= DAV_ERR_RECV_PROTOCOL;

				(* Timeout *)
				ELSIF(TON_10ms_Timeout.Q)THEN
					status:= DAV_ERR_TIMEOUT;

				(* Error *)
				ELSIF(DAVmpiRead_0.status <> 65535)THEN
					status:= DAVmpiRead_0.status;
				END_IF
			(**************************************************************************************************************************)

			(**************************************************************************************************************************)
			(* MPI Read - STX					                                                               																	*)
			(**************************************************************************************************************************)
			204:
				(* Service function *)
        DAVmpiRead_0();

				(* Service timeout *)
				TON_10ms_Timeout();

				(* Data received *)
				IF((DAVmpiRead_0.status = 0) AND (DAVmpiRead_0.recvBufferLength = 1) AND (bufferRead[0] = 16#02))THEN

					(* Reset timer *)
					TON_10ms_Timeout.IN:= FALSE;
					TON_10ms_Timeout();
					TON_10ms_Timeout.IN:= TRUE;

					(* Create message to send *)
					bufferSend[0]:= 						16#10;								(* DLE *)
					DAVmpiSend_0.sendLength:=		1;										(* Length to send *)

					(* Continue *)
					bufferRead[0]:= 0;
					state:= 205;

				(* Invalid protocol *)
				ELSIF(DAVmpiRead_0.status = 0)THEN
					status:= DAV_ERR_RECV_PROTOCOL;

				(* Timeout *)
				ELSIF(TON_10ms_Timeout.Q)THEN
					status:= DAV_ERR_TIMEOUT;

				(* Error *)
				ELSIF(DAVmpiRead_0.status <> 65535)THEN
					status:= DAVmpiRead_0.status;
				END_IF
			(**************************************************************************************************************************)

			(**************************************************************************************************************************)
			(* MPI Write - DLE		                                                                   																	*)
			(**************************************************************************************************************************)
			205:
				(* Service function *)
				DAVmpiSend_0();

				(* Data written *)
				IF(DAVmpiSend_0.status = 0)THEN

					(* Point to the message buffer *)
					IF(mpiFullExchange = FALSE)THEN
						DAVmpiRead_0.pBufferR:=			pDAV.pBufferR;
						DAVmpiRead_0.readLength:=		DAV_DEFAULT_BUFFER_R;
 					END_IF

					(* Continue *)
					bufferSend[0]:= 0;
					state:= 206;

				(* Error writing data *)
				ELSIF(DAVmpiSend_0.status <> 65535)THEN
					status:= DAVmpiSend_0.status;
				END_IF
			(**************************************************************************************************************************)

			(**************************************************************************************************************************)
			(* MPI Read - message / ack			                                                         																	*)
			(**************************************************************************************************************************)
			206:
				(* Service function *)
	      DAVmpiRead_0();

				(* Service timeout *)
				TON_10ms_Timeout();

				(* Data received *)
				IF((DAVmpiRead_0.status = 0) AND (DAVmpiRead_0.recvBufferLength > 0))THEN

					(* Reset timer *)
					TON_10ms_Timeout.IN:= FALSE;
					TON_10ms_Timeout();
					TON_10ms_Timeout.IN:= TRUE;

					(* Point to the internal buffer *)
					DAVmpiRead_0.pBufferR:=			ADR(bufferRead);
					DAVmpiRead_0.readLength:=		SIZEOF(bufferRead);

					(* Create message to send *)
					bufferSend[0]:= 						16#10;									(* DLE *)
					DAVmpiSend_0.sendLength:=		1;

		 			(* Return received length *)
					IF(mpiFullExchange = FALSE)THEN
						recvLength:= DAVmpiRead_0.recvBufferLength;
					END_IF
					state:= 207;

				(* Invalid protocol *)
				ELSIF(DAVmpiRead_0.status = 0)THEN
					status:= DAV_ERR_RECV_PROTOCOL;

				(* Timeout *)
				ELSIF(TON_10ms_Timeout.Q)THEN
					status:= DAV_ERR_TIMEOUT;

				(* Error *)
				ELSIF(DAVmpiRead_0.status <> 65535)THEN
					status:= DAVmpiRead_0.status;
				END_IF
			(**************************************************************************************************************************)

			(**************************************************************************************************************************)
			(* MPI Write - DLE		                                                                   																	*)
			(**************************************************************************************************************************)
			207:
				(* Service function *)
				DAVmpiSend_0();

				(* Data written *)
				IF(DAVmpiSend_0.status = 0)THEN
					bufferSend[0]:= 0;

					(* Complete *)
					IF(mpiFullExchange = FALSE)THEN
						status:= 0;

					(* Check for a valid ACK *)
					(*	1) Length is 12 *)
					(*	2) Position 6 contains 16#B0 - used for an acknowledge *)
					(*	3) Position 8 contains the required acknowledge number *)
					ELSE

						(* Remove DLE doubling *)
						recvLength:= DAVdecodeMPI(ADR(bufferRead), SIZEOF(bufferRead), DAVmpiRead_0.recvBufferLength);
						IF((recvLength = 12) AND (bufferRead[6] = 16#B0) AND (bufferRead[8] = pDAV.connection.ackNum))THEN

							(* Store acknowledge number to send *)
							sendAckNumber:= bufferRead[7];
							memset(ADR(bufferRead), 0, SIZEOF(bufferRead));
							state:= 208;

						(* Invalid ACK packet *)
						ELSE
			 				status:= DAV_ERR_ACKNOWLEDGE;
						END_IF
					END_IF

				(* Error writing data *)
				ELSIF(DAVmpiSend_0.status <> 65535)THEN
					status:= DAVmpiSend_0.status;
				END_IF
			(**************************************************************************************************************************)

			(**************************************************************************************************************************)
			(* MPI Read - STX					                                                               																	*)
			(**************************************************************************************************************************)
			208:
				(* Service function *)
        DAVmpiRead_0();

				(* Service timeout *)
				TON_10ms_Timeout();

				(* Data received *)
				IF((DAVmpiRead_0.status = 0) AND (DAVmpiRead_0.recvBufferLength = 1) AND (bufferRead[0] = 16#02))THEN

					(* Reset timer *)
					TON_10ms_Timeout.IN:= FALSE;
					TON_10ms_Timeout();
					TON_10ms_Timeout.IN:= TRUE;

					(* Create message to send *)
					bufferSend[0]:= 						16#10;								(* DLE *)
					DAVmpiSend_0.sendLength:=		1;										(* Length to send *)

					(* Continue *)
					bufferRead[0]:= 0;
					state:= 209;

				(* Invalid protocol *)
				ELSIF(DAVmpiRead_0.status = 0)THEN
					status:= DAV_ERR_RECV_PROTOCOL;

				(* Timeout *)
				ELSIF(TON_10ms_Timeout.Q)THEN
					status:= DAV_ERR_TIMEOUT;

				(* Error *)
				ELSIF(DAVmpiRead_0.status <> 65535)THEN
					status:= DAVmpiRead_0.status;
				END_IF
			(**************************************************************************************************************************)

			(**************************************************************************************************************************)
			(* MPI Write - DLE		                                                                   																	*)
			(**************************************************************************************************************************)
			209:
				(* Service function *)
				DAVmpiSend_0();

				(* Data written *)
				IF(DAVmpiSend_0.status = 0)THEN

					(* Point to the message buffer *)
					memset(pDAV.pBufferR, 0, DAV_DEFAULT_BUFFER_R);
					DAVmpiRead_0.pBufferR:=			pDAV.pBufferR;
					DAVmpiRead_0.readLength:=		DAV_DEFAULT_BUFFER_R;

					(* Continue *)
					bufferSend[0]:= 0;
					state:= 210;

				(* Error writing data *)
				ELSIF(DAVmpiSend_0.status <> 65535)THEN
					status:= DAVmpiSend_0.status;
				END_IF
			(**************************************************************************************************************************)

			(**************************************************************************************************************************)
			(* MPI Read - message			                                                         																						*)
			(**************************************************************************************************************************)
			210:
				(* Service function *)
	      DAVmpiRead_0();

				(* Service timeout *)
				TON_10ms_Timeout();

				(* Data received *)
				IF((DAVmpiRead_0.status = 0) AND (DAVmpiRead_0.recvBufferLength > 0))THEN

					(* Reset timer *)
					TON_10ms_Timeout.IN:= FALSE;
					TON_10ms_Timeout();
					TON_10ms_Timeout.IN:= TRUE;

					(* Point to the internal buffer *)
					DAVmpiRead_0.pBufferR:=			ADR(bufferRead);
					DAVmpiRead_0.readLength:=		SIZEOF(bufferRead);

					(* Create message to send *)
					bufferSend[0]:= 						16#10;									(* DLE *)
					DAVmpiSend_0.sendLength:=		1;

					(* Store acknowledge number to send *)
					sendAckNumber:= ppBuffer[7];

					(* Return received length *)
					recvLength:= DAVmpiRead_0.recvBufferLength;
					state:= 211;

				(* Invalid protocol *)
				ELSIF(DAVmpiRead_0.status = 0)THEN
					status:= DAV_ERR_RECV_PROTOCOL;

				(* Timeout *)
				ELSIF(TON_10ms_Timeout.Q)THEN
					status:= DAV_ERR_TIMEOUT;

				(* Error *)
				ELSIF(DAVmpiRead_0.status <> 65535)THEN
					status:= DAVmpiRead_0.status;
				END_IF
			(**************************************************************************************************************************)

			(**************************************************************************************************************************)
			(* MPI Write - DLE			                                                                 																	*)
			(**************************************************************************************************************************)
			211:
				(* Service function *)
				DAVmpiSend_0();

				(* Data written *)
				IF(DAVmpiSend_0.status = 0)THEN

					(* Create message to send *)
					bufferSend[0]:= 						16#02;									(* STX *)
					DAVmpiSend_0.sendLength:=		1;
					state:= 212;

				(* Error writing data *)
				ELSIF(DAVmpiSend_0.status <> 65535)THEN
					status:= DAVmpiSend_0.status;
				END_IF
			(**************************************************************************************************************************)

			(**************************************************************************************************************************)
			(* MPI Write - STX                                                                  																			*)
			(**************************************************************************************************************************)
			212:
				(* Service function *)
				DAVmpiSend_0();

				(* Data written *)
				IF(DAVmpiSend_0.status = 0)THEN

					(* Continue *)
					bufferSend[0]:= 0;
					state:= 213;

				(* Error writing data *)
				ELSIF(DAVmpiSend_0.status <> 65535)THEN
					status:= DAVmpiSend_0.status;
				END_IF
			(**************************************************************************************************************************)

			(**************************************************************************************************************************)
			(* MPI Read - DLE                                                               																					*)
			(**************************************************************************************************************************)
			213:
				(* Service function *)
        DAVmpiRead_0();

				(* Service timeout *)
				TON_10ms_Timeout();

				(* Data received *)
				IF((DAVmpiRead_0.status = 0) AND (DAVmpiRead_0.recvBufferLength = 1) AND (bufferRead[0] = 16#10))THEN

					(* Reset timer *)
					TON_10ms_Timeout.IN:= FALSE;
					TON_10ms_Timeout();
					TON_10ms_Timeout.IN:= TRUE;

					(* Create message to send *)
					DAVmpiSend_0.sendLength:= DAVpacketMPIack(ADR(pDAV), ADR(bufferSend), sendAckNumber);

		 			(* Continue *)
					bufferRead[0]:= 0;
	 				state:= 214;

				(* Invalid protocol *)
				ELSIF(DAVmpiRead_0.status = 0)THEN
					status:= DAV_ERR_RECV_PROTOCOL;

				(* Timeout *)
				ELSIF(TON_10ms_Timeout.Q)THEN
					status:= DAV_ERR_TIMEOUT;

				(* Error *)
				ELSIF(DAVmpiRead_0.status <> 65535)THEN
					status:= DAVmpiRead_0.status;
				END_IF
			(**************************************************************************************************************************)

			(**************************************************************************************************************************)
			(* MPI Write - ack		                                                                   																	*)
			(**************************************************************************************************************************)
			214:
				(* Service function *)
				DAVmpiSend_0();

				(* Data written *)
				IF(DAVmpiSend_0.status = 0)THEN
					memset(ADR(bufferSend), 0, SIZEOF(bufferSend));
			 		state:= 215;

				(* Error writing data *)
				ELSIF(DAVmpiSend_0.status <> 65535)THEN
					status:= DAVmpiSend_0.status;
				END_IF
			(**************************************************************************************************************************)

			(**************************************************************************************************************************)
			(* MPI Read - DLE                                                               																					*)
			(**************************************************************************************************************************)
			215:
				(* Service function *)
        DAVmpiRead_0();

				(* Service timeout *)
				TON_10ms_Timeout();

				(* Data received *)
				IF((DAVmpiRead_0.status = 0) AND (DAVmpiRead_0.recvBufferLength = 1) AND (bufferRead[0] = 16#10))THEN

					(* Reset timer *)
					TON_10ms_Timeout.IN:= FALSE;
					TON_10ms_Timeout();
					TON_10ms_Timeout.IN:= TRUE;

		 			(* Internal *)
					bufferRead[0]:= 0;
					status:= 0;

					(* Remove DLE doubling *)
					recvLength:= DAVdecodeMPI(pDAV.pBufferR, DAV_DEFAULT_BUFFER_R, recvLength);

					(* Return Parameter and Data lengths *)
					recvParamLength:= DAVswapWORD(ADR(ppBuffer[14]));				(* Bytes ppBuffer[14] and [15] *)
					recvDataLength:= DAVswapWORD(ADR(ppBuffer[16]));				(* Bytes ppBuffer[16] and [17] *)

					(* Return the start of the data index *)
					IF((ppBuffer[9] = 2) OR (ppBuffer[9] = 3))THEN
						recvStartOfDataIdx:= 20; (*8 + 12;*)
					ELSE
						recvStartOfDataIdx:= 18; (*8 + 10;*)
					END_IF

					(* Reduce receive length for length of data *)
					IF(recvLength >= recvStartOfDataIdx)THEN
		 				recvLength:= recvLength - recvStartOfDataIdx;
					ELSE
						recvLength:= 0;
					END_IF

				(* Invalid protocol *)
				ELSIF(DAVmpiRead_0.status = 0)THEN
					status:= DAV_ERR_RECV_PROTOCOL;

				(* Timeout *)
				ELSIF(TON_10ms_Timeout.Q)THEN
					status:= DAV_ERR_TIMEOUT;

				(* Error *)
				ELSIF(DAVmpiRead_0.status <> 65535)THEN
					status:= DAVmpiRead_0.status;
				END_IF
			(**************************************************************************************************************************)

		END_CASE
		(****************************************************************************************************************************)
		(* End of Function Operation                                                              																	*)
		(****************************************************************************************************************************)

		(****************************************************************************************************************************)
		(* Reset to state 0 when complete	(or in error)																																							*)
		(****************************************************************************************************************************)
		IF(status <> 65535)THEN
			lastState:= state;
			state:= 0;
		END_IF
		(****************************************************************************************************************************)

	END_IF
END_FUNCTION_BLOCK
(********************************************************************************************************************************)
(* End of DAVsend																																																								*)
(********************************************************************************************************************************)

(********************************************************************************************************************************)
(* DAVmpiSend																																																										*)
(*==============================================================================================================================*)
(* Write data to a Siemen's PLC			 																																														*)
(* Returns a status																																																							*)
(********************************************************************************************************************************)
FUNCTION_BLOCK DAVmpiSend

	(* Function not enabled *)
	IF(enable = FALSE)THEN
		status:= 65534;

	(* Invalid buffer pointer *)
	ELSIF(pBufferW = 0)THEN
 		status:= DAV_ERR_BUFFER;

	(* Invalid length *)
	ELSIF(sendLength = 0)THEN
 		status:= DAV_ERR_SEND_NODATA;

	(* Run the function *)
	ELSE

		(* Make function status busy *)
		status:= 65535;

		(* Service function *)
		FRM_gbuf_0.enable:=					TRUE;										(* Enable function block *)
		FRM_gbuf_0.ident:=					ident;									(* FRM_Xopen ident *)
		FRM_gbuf_0();

		(* Buffer available *)
		IF((FRM_gbuf_0.status = 0) AND (FRM_gbuf_0.buffer <> 0) AND (FRM_gbuf_0.buflng >= sendLength))THEN

			(* Store data to write *)
			IF(FRM_gbuf_0.buflng > sendLength)THEN
				memcpy(FRM_gbuf_0.buffer, pBufferW, sendLength);
			ELSE
				memcpy(FRM_gbuf_0.buffer, pBufferW, FRM_gbuf_0.buflng);
			END_IF

			(* Service function *)
			FRM_write_0.enable:=			TRUE;										(* Enable function block *)
			FRM_write_0.ident:=				ident;									(* FRM_Xopen ident *)
			FRM_write_0.buffer:=			FRM_gbuf_0.buffer;			(* Write buffer *)
			FRM_write_0.buflng:= 			sendLength;							(* Write buffer length *)
			FRM_write_0();																		(* Service the function block *)

			(* Data written *)
			IF(FRM_write_0.status = 0)THEN
				status:= 0;

			(* Error writing data *)
			ELSE
				status:= FRM_write_0.status;

				(* Manually release buffer *)
				FRM_robuf_0.enable:= 		TRUE;										(* Enable function block *)
				FRM_robuf_0.ident:=			ident;									(* FRM_Xopen ident *)
				FRM_robuf_0.buffer:=		FRM_gbuf_0.buffer;			(* Write buffer *)
				FRM_robuf_0.buflng:=		FRM_gbuf_0.buflng;			(* Write buffer length *)
				FRM_robuf_0();
			END_IF

		(* Buffer not large enough *)
		ELSIF(FRM_gbuf_0.status = 0)THEN
			status:= DAV_ERR_SEND_BUFFERSIZE;

		(* Error *)
		ELSIF(FRM_gbuf_0.status <> 65535)THEN
			status:= FRM_gbuf_0.status;
		END_IF
	END_IF
END_FUNCTION_BLOCK
(********************************************************************************************************************************)
(* End of DAVmpiSend																																																						*)
(********************************************************************************************************************************)

(********************************************************************************************************************************)
(* DAVmpiRead																																																										*)
(*==============================================================================================================================*)
(* Reads data to a Siemen's PLC			 																																														*)
(* Returns a status																																																							*)
(********************************************************************************************************************************)
FUNCTION_BLOCK DAVmpiRead

	(* Clear received buffer length *)
	recvBufferLength:= 0;

	(* Function not enabled *)
	IF(enable = FALSE)THEN
		status:= 65534;

	(* Invalid buffer pointer *)
	ELSIF(pBufferR = 0)THEN
 		status:= DAV_ERR_BUFFER;

	(* Invalid length *)
	ELSIF(readLength = 0)THEN
 		status:= DAV_ERR_BUFFER_SIZE;

	(* Run the function *)
	ELSE

		(* Make function status busy *)
		status:= 65535;

		(* Service function *)
		FRM_read_0.enable:=			TRUE;										(* Enable function block *)
		FRM_read_0.ident:=			ident;									(* FRM_Xopen ident *)
 		FRM_read_0();

		(* Data received *)
		IF((FRM_read_0.status = 0) AND (FRM_read_0.buflng > 0) AND (FRM_read_0.buffer <> 0))THEN

			(* Copy data *)
			IF(FRM_read_0.buflng <= readLength)THEN
				memset(pBufferR, 0, readLength);						(* Clear data *)
				memcpy(pBufferR, FRM_read_0.buffer, FRM_read_0.buflng);
				recvBufferLength:= FRM_read_0.buflng;				(* Buffer length *)

			(* Buffer too small *)
			ELSE
				status:= DAV_ERR_RECV_BUFFERSIZE;
			END_IF

			(* Release the read buffer *)
			FRM_rbuf_0.enable:=		TRUE;										(* Read buffer *)
			FRM_rbuf_0.ident:=		ident;									(* Read buffer length *)
			FRM_rbuf_0.buffer:= 	FRM_read_0.buffer;			(* Read buffer *)
			FRM_rbuf_0.buflng:= 	FRM_read_0.buflng;			(* Read buffer length *)
			FRM_rbuf_0();																	(* Service the function block *)

			(* Buffer released *)
			IF(FRM_rbuf_0.status <> 0)THEN
				status:= FRM_rbuf_0.status;

			(* Function complete *)
			ELSIF(status = 65535)THEN
				status:= 0;
			END_IF

		(* Invalid receive length *)
		ELSIF(FRM_read_0.status = 0)THEN
			status:= DAV_ERR_RECV_NODATA;

		(* No data - try again *)
		ELSIF(FRM_read_0.status = frmERR_NOINPUT)THEN
			status:= 65535;

		(* Error *)
		ELSIF(FRM_read_0.status <> 65535)THEN
			status:= FRM_read_0.status;
		END_IF
	END_IF
END_FUNCTION_BLOCK
(********************************************************************************************************************************)
(* End of DAVmpiRead																																																						*)
(********************************************************************************************************************************)
```
